Fanuc KAREL source: kt00258.KL

PROGRAM KT00258
%STACKSIZE=65535
%PRIORITY=65535
%NOLOCKGROUP
VAR
I1 : INTEGER
R2 : REAL
OUT : BOOLEAN
BEGIN
I1=2
R2=3.0
OUT=(R2=(I1))
END KT00258
